(* IEC 61131-3 sources: repolevel_ST_code_completion/output/0122完整版本_无planner目前sota/repoeval_PID_controller/readful_result_no_provide, 4 files *)

(* ---- HeatExchanger.st ---- *)
VAR
	now: TIME;
	lastTime: TIME;
	lastPV: REAL := 140;
	A: REAL;
	B: REAL;
	delta_t: REAL;
	deadTimeElapsed: TIME := T#0ms;
END_VAR
VAR CONSTANT
	millis: REAL := 1000;
END_VAR

now := TIME();
IF ((now - lastTime) > Sample_time) THEN
	delta_t := TIME_TO_REAL(Sample_time) / millis;
	A := EXP(-delta_t / Tp);
	B := 1 - A;

IF (deadTimeElapsed >= REAL_TO_TIME(Dead_t)) THEN
    PV := A * lastPV + B * Kp * CO + C;
    lastPV := PV;
  ELSE
    deadTimeElapsed := deadTimeElapsed + Sample_time;
  END_IF;

	lastTime := now;
END_IF;
END_FUNCTION_BLOCK

(* ---- HeatExchanger2.st ---- *)
VAR
	now: TIME;
	lastTime: TIME := T#0s;
	delta_t: REAL;
	heat_flow: REAL;
	lastTemp: REAL;
END_VAR
VAR CONSTANT
	millis: REAL := 1000;
END_VAR

now := TIME();
IF ((now - lastTime) > Sample_time) THEN
// Convert TIME to REAL for arithmetic operation
  delta_t := TIME_TO_REAL(now - lastTime) / millis;
	heat_flow := Heat_In + U * (Temp_Out - Temp_In);
	Temp := Temp_In + (heat_flow * delta_t / TC);
	lastTime := now;
END_IF;
RETURN;
END_FUNCTION_BLOCK

(* ---- PID_controller.st ---- *)
VAR
	lastErr: REAL := 0; //Previous error
	integral: REAL := 0; //Integral accumulator
	deltaTime: REAL := 0; //Time difference
	deltaPV: REAL := 0; //Change in process variable
END_VAR

// Handle time and error calculation via existing logic only
// Adjust computations dependent on undefined variables
deltaTime := TO_REAL(SampleTime) / TO_REAL(millis); //Proper type conversion for calculation

// Proportional term
CO_P := Kc * (SP - PV);

// Integral term with anti-windup
integral := integral + ((SP - PV) * deltaTime);
IF integral > UpperLimit THEN
  integral := UpperLimit;
ELSIF integral < LowerLimit THEN
  integral := LowerLimit;
END_IF;
CO_I := Kc * (integral / Ti);

// Derivative term
CO_D := -Kc * (Td * (PV - lastErr) / deltaTime);

// Calculate total controller output
CO := CO_P + CO_I + CO_D;

// Apply output limits
IF CO > UpperLimit THEN
  CO := UpperLimit;
ELSIF CO < LowerLimit THEN
  CO := LowerLimit;
END_IF;

// Update last values
lastErr := PV;
// Variable `lastTime` is undefined; its update is removed
END_FUNCTION_BLOCK

(* ---- Tank.st ---- *)
VAR
	now: TIME;
	lastTime: TIME := T#0ms;
	proc_sum_in: REAL := 0.0;
	proc_sum_out: REAL := 0.0;
	temp: REAL := 0.0;
	millis: UINT := 1000;
	proc_out: REAL := 0.0;
END_VAR

now := TIME();
IF (now - lastTime) >= SampleTime THEN
	// Update the fluid level based on input and output flow rates
	Level := Level + TIME_TO_REAL(SampleTime) / millis * (Process_In - Process_Out);

	// Ensure the level does not exceed the defined limits
	IF Level < Lower_limit THEN
		Level := Lower_limit;
	ELSIF Level > Upper_limit THEN
		Level := Upper_limit;
	END_IF;

	// Update the last time variable
	lastTime := now;
END_IF;
END_FUNCTION_BLOCK
